FUNCTION_BLOCK EVENTS_PRIOITY_OR (* Basic Function Block Type *)
  (* Standard: 61499-2 *)
  (* Version 0.0, 6/26/2018, Eskimos, nxtControl GmbH, Template *)
  PACKAGE Main;
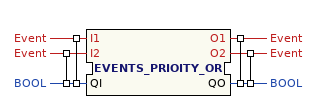
  EVENT_INPUT
    I1 WITH QI; (* Higher Priority *)
    I2 WITH QI; (* Lower priority *)
  END_EVENT
  EVENT_OUTPUT
    O1 WITH QO; (* Higher Prioity *)
    O2 WITH QO; (* Lower priority *)
  END_EVENT
  VAR_INPUT
    QI : BOOL; (* Input event qualifier *)
  END_VAR
  VAR_OUTPUT
    QO : BOOL; (* Output event qualifier *)
  END_VAR
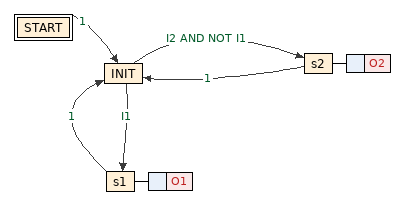
  EC_STATES
    START; (* Initial State *)
    s1 : -> O1; (* Normal execution *)
    s2 : -> O2;
    INIT;
  END_STATES
  EC_TRANSITIONS
    INIT TO s1 := I1;
    s1 TO INIT := 1;
    INIT TO s2 := I2 AND NOT I1;
    s2 TO INIT := 1;
    START TO INIT := 1;
  END_TRANSITIONS
END_FUNCTION_BLOCK
